(* Logix 5000 project; controller lab_1 vendor 1 type 14 code 96 rev 28.11; software revision 28.00 *)

TASK MainTask (continuous, watchdog 500 ms) : MainProgram

MODULES
   Local : vendor 1 type 14 code 96 (ICP 1, rev 28.11)
      INPUT : vendor 1 type 7 code 2 (ICP 2, rev 3.1, Input RPI 20 ms)
      RELAY_4 : 1756-OW16I (ICP 4, rev 3.1, Output RPI 20 ms)
      Relay_1 : 1756-OW16I (ICP 0, rev 3.3, Output RPI 20 ms)
      Relay_8 : 1756-IF6I (ICP 8, rev 1.1, Input RPI 100 ms)
      Relay_7 : vendor 1 type 10 code 4 (ICP 7, rev 1.12, Output RPI 25 ms)
      enet : vendor 1 type 12 code 219 (ICP 9, Ethernet 192.168.1.7, rev 10.1)
         REMOTE_IO : 1734-AENTR (Ethernet 192.168.1.10, rev 5.1, Output RPI 20 ms)
            input_1 : vendor 1 type 7 code 307 (PointIO 1, rev 3.1)
            input_2 : vendor 1 type 7 code 307 (PointIO 2, rev 3.1)
            input_3 : vendor 1 type 7 code 307 (PointIO 3, rev 3.1)
            input_4 : vendor 1 type 7 code 307 (PointIO 4, rev 3.1)
            output5 : vendor 1 type 7 code 134 (PointIO 5, rev 3.1)
            output6 : vendor 1 type 7 code 134 (PointIO 6, rev 3.1)
            output7 : vendor 1 type 7 code 134 (PointIO 7, rev 3.1)
END_MODULES

PROGRAM MainProgram   (* main routine MainRoutine *)
VAR
   ADD : BOOL;
   ALARM : ALIAS FOR REMOTE_IO:2:I.0;
   BAND_01 : FBD_BOOLEAN_AND := (In1 := 1, In2 := 1, In3 := 1, In4 := 1, In5 := 1, In6 := 1, In7 := 1, In8 := 1);
   BNOT_01 : FBD_BOOLEAN_NOT := (Out := 1);
   BNOT_02 : FBD_BOOLEAN_NOT := (Out := 1);
   BOR_01 : FBD_BOOLEAN_OR;
   ESTOP : ALIAS FOR Local:2:I.Data.8;
   FLASHER : BOOL := 1;
   GREEN_LIGHT : ALIAS FOR Local:4:O.Data.3;
   Meter_0 : ALIAS FOR Local:7:O.Ch0Data;
   Meter_1 : ALIAS FOR Local:7:O.Ch1Data;
   OFF_TIMER : TIMER := (PRE := 5000);
   ON_TIMER : TIMER := (PRE := 5000, EN := 1, TT := 1);
   POT_0 : ALIAS FOR Local:8:I.Ch0Data;
   POT_1 : ALIAS FOR Local:8:I.Ch1Data;
   RED_LIGHT : ALIAS FOR Local:4:O.Data.2;
   run : BOOL;
   RUN_CMD : BOOL;
   START : ALIAS FOR Local:2:I.Data.0;
   STOP : ALIAS FOR Local:2:I.Data.9;
   time_off : DINT := 5000;
   time_on : DINT := 5000;
   TONR_01 : FBD_TIMER := (TimerEnable := 1, PRE := 2000, ACC := 2000, EN := 1, DN := 1);
   TONR_02 : FBD_TIMER := (TimerEnable := 1, PRE := 2000, ACC := 796, EN := 1, TT := 1);
   YELLOW_LIGHT : ALIAS FOR Local:4:O.Data.1;
END_VAR

ROUTINE ADD_IT2_LD   (* ladder *)
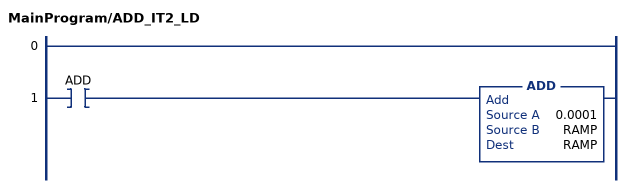
   0: ;
   1: XIC(ADD)ADD(0.0001,RAMP,RAMP);
END_ROUTINE

ROUTINE ADD_IT_LD   (* ladder *)
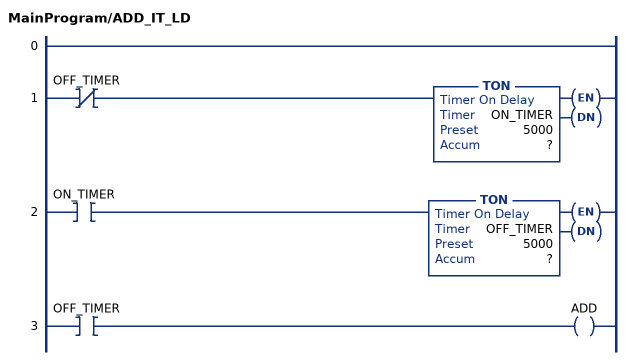
   0: ;
   1: XIO(OFF_TIMER)TON(ON_TIMER,?,?);
   2: XIC(ON_TIMER)TON(OFF_TIMER,?,?);
   3: XIC(OFF_TIMER)OTE(ADD);
END_ROUTINE

ROUTINE ANALOG_COMPARE   (* ladder *)
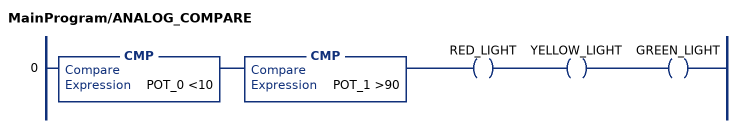
   0: CMP(POT_0 <10)CMP(POT_1 >90)OTE(RED_LIGHT)OTE(YELLOW_LIGHT)OTE(GREEN_LIGHT);
END_ROUTINE

ROUTINE ANALOG_COMPUTE   (* ladder *)
   0: ;
END_ROUTINE

ROUTINE ANALOG_LESS_AND_GREAT   (* ladder *)
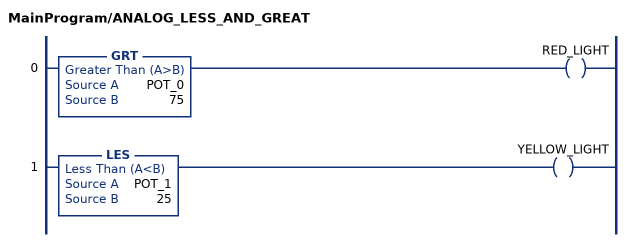
   0: GRT(POT_0,75)OTE(RED_LIGHT);
   1: LES(POT_1,25)OTE(YELLOW_LIGHT);
END_ROUTINE

ROUTINE ANALOG_LIMIT   (* ladder *)
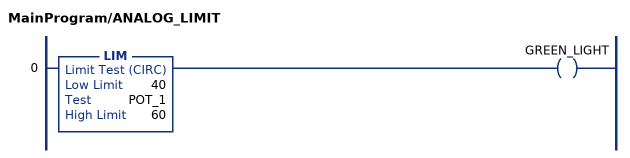
   0: LIM(40,POT_1,60)OTE(GREEN_LIGHT);
END_ROUTINE

ROUTINE ANALOG_METER   (* ladder *)
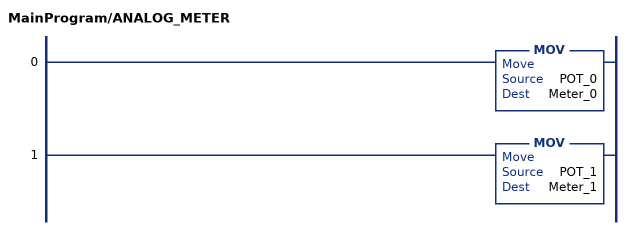
   0: MOV(POT_0,Meter_0);
   1: MOV(POT_1,Meter_1);
END_ROUTINE

ROUTINE FBD_Motor_Control   (* function block diagram *)
   SHEET 1
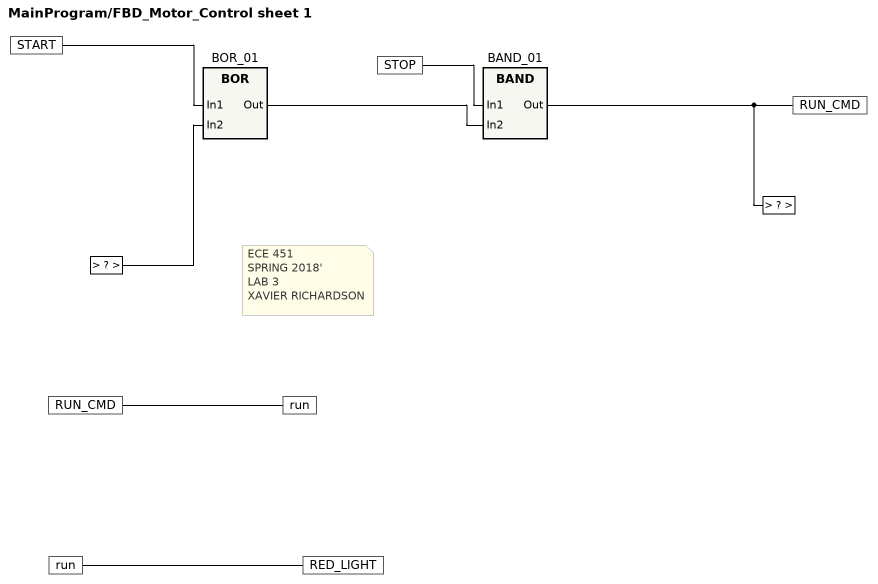
   // ECE 451
   // SPRING 2018'
   // LAB 3
   // XAVIER RICHARDSON
   BOR_01 : BOR(In1 := START, In2 := WIRE(?) {feedback});
   run := RUN_CMD;
   RED_LIGHT := run;
   BAND_01 : BAND(In1 := STOP, In2 := BOR_01.Out);
   WIRE(?) := BAND_01.Out;
   RUN_CMD := BAND_01.Out;
END_ROUTINE

ROUTINE FLASHER_FD   (* function block diagram *)
   SHEET 1
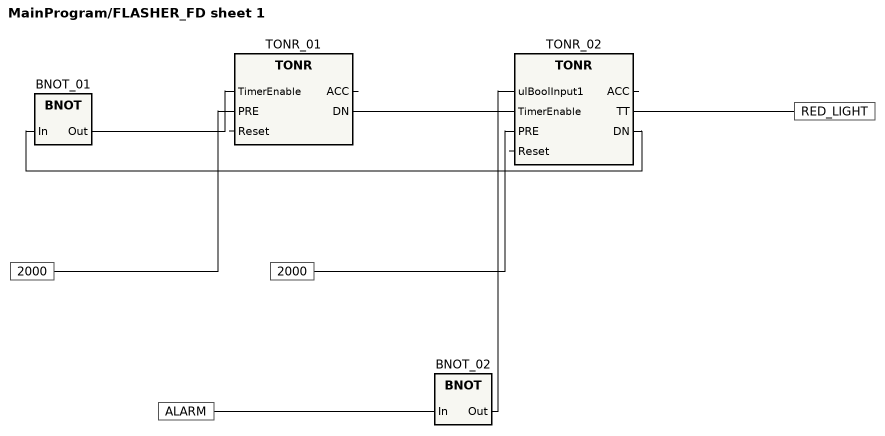
   BNOT_01 : BNOT(In := TONR_02.DN {feedback});
   TONR_01 : TONR(TimerEnable := BNOT_01.Out, PRE := 2000);   // unwired pins: Reset ACC
   BNOT_02 : BNOT(In := ALARM);
   TONR_02 : TONR(ulBoolInput1 := BNOT_02.Out, TimerEnable := TONR_01.DN, PRE := 2000);   // unwired pins: Reset ACC
   RED_LIGHT := TONR_02.TT;
END_ROUTINE

ROUTINE FLASHER_L   (* ladder *)
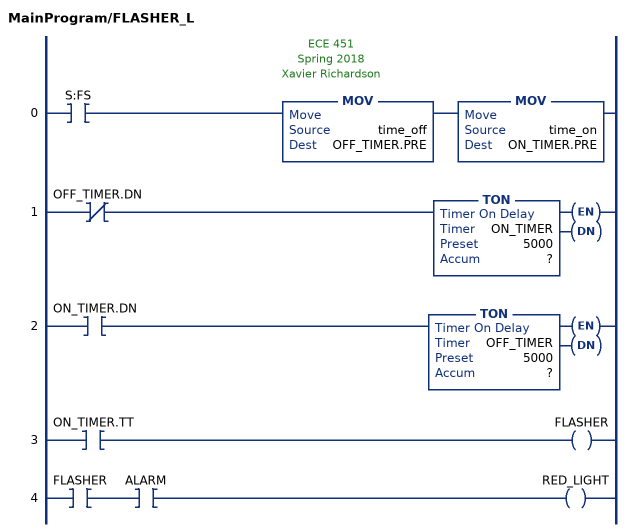
   // ECE 451
   // Spring 2018
   // Xavier Richardson
   0: XIC(S:FS)MOV(time_off,OFF_TIMER.PRE)MOV(time_on,ON_TIMER.PRE);
   1: XIO(OFF_TIMER.DN)TON(ON_TIMER,?,?);
   2: XIC(ON_TIMER.DN)TON(OFF_TIMER,?,?);
   3: XIC(ON_TIMER.TT)OTE(FLASHER);
   4: XIC(FLASHER)XIC(ALARM)OTE(RED_LIGHT);
END_ROUTINE

ROUTINE FLASHER_ST   (* structured text *)
   TONR_01.PRE := 2000;
   
   TONR_01.TimerEnable := NOT TONR_02.DN;
   
   TONR(TONR_01);
   
   
   /////////////////////////////////////////////
   TONR_02.PRE := 2000;
   
   TONR_02.TimerEnable := TONR_01.DN;
   
   TONR_02.EnableIn := NOT ALARM;
   
   TONR(TONR_02);
   
   /////////////////////////////////////////////
   
   RED_LIGHT:= TONR_02.TT;
   
   
   
END_ROUTINE

ROUTINE MainRoutine   (* ladder *)
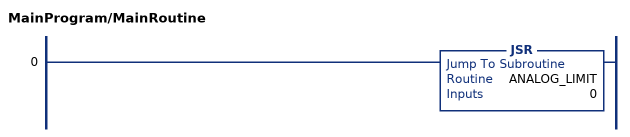
   0: JSR(ANALOG_LIMIT,0);
END_ROUTINE

ROUTINE ST_Motor_Control   (* structured text *)
   (*
   ECE 451 SPRING 2018
   XAVIER RICHARDSON
   *)
   
   //1ST RUNG
   
   RUN_CMD := (START or RUN_CMD) and STOP AND ESTOP;
   
   /////2ND RUNG
   
   run := RUN_CMD;
   
   ////////////3RD RUNG
   
   run := RED_LIGHT;
END_ROUTINE
END_PROGRAM
